FUNCTION_BLOCK PUBLIC FINAL ConcreteADSLogger EXTENDS AbstractLogger
VAR_INPUT
END_VAR
VAR_OUTPUT
END_VAR
VAR
END_VAR

METHOD PROTECTED InternalLog
VAR_INPUT
     Message:STRING;
END_VAR
_Busy:=TRUE;
 
ADSLOGSTR(    msgCtrlMask:=ADSLOG_MSGTYPE_LOG,
              msgFmtStr:=Message,
              strArg:='');
             
_Busy:=FALSE;
END_METHOD

END_FUNCTION_BLOCK

(* stored: Version 1.1.0.1, ProductVersion 3.1.4024.12
   POU ConcreteADSLogger: Id {bcd41922-23fa-4c27-9719-0a03add0316b}, SpecialFunc None
   Method InternalLog: Id {e1dbd88f-0eb2-4e8b-9585-69e7edd4ab47} *)
